PROGRAM MAIN_FBD_IL_LD //use menu "FBD/IL/LD" to switch language between FBD, IL and LD offline or online 
VAR
	Timer					: TON;
	fbFBD_IL_LD_SamplePOU 	: FB_FBD_IL_LD_SamplePOU;

	eOperation		: E_Operation := eOp_Add;
	eOperationPrev	: E_Operation := eOp_Add;
	iResultC		: DINT;
	bZero			: BOOL;
	bPos			: BOOL;
	bNeg			: BOOL;
	bTest			: BOOL;
	tTimerValue		: TIME := T#3S;
END_VAR
VAR // added by the converter: edge detectors and wires of the graphical bodies
    _w1, _w2, _w3 : ANY;
END_VAR

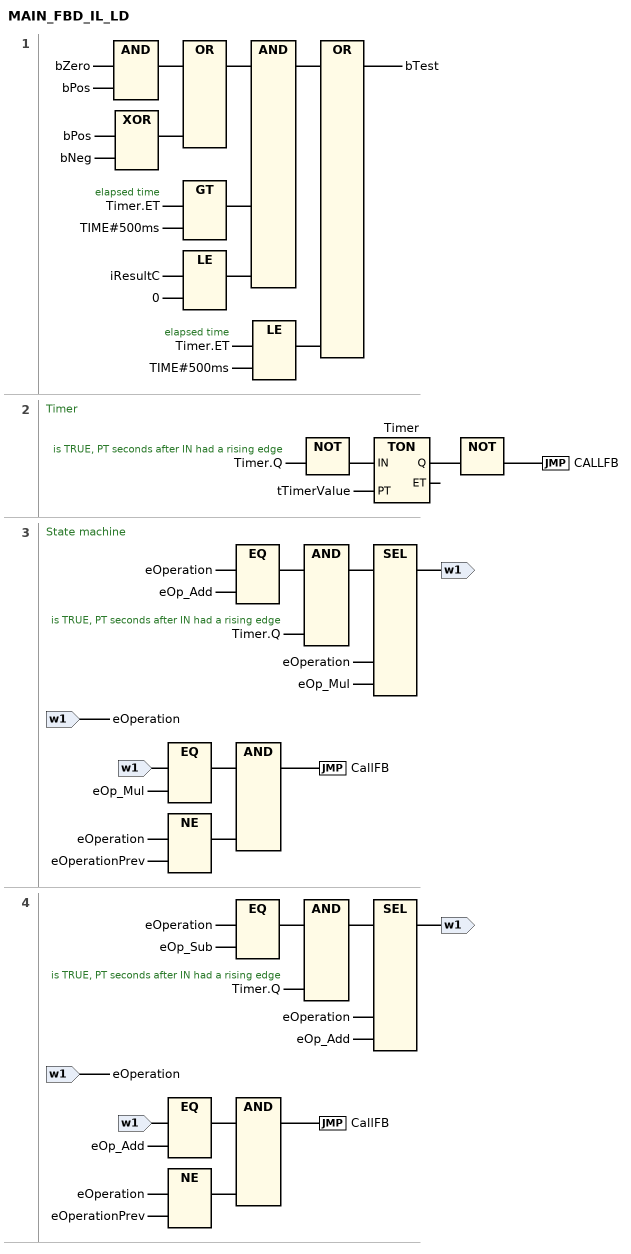
// NETWORK 1
//   Timer.ET: elapsed time
bTest := (bZero AND bPos OR bPos XOR bNeg) AND Timer.ET > TIME#500ms AND iResultC <= 0 OR Timer.ET <= TIME#500ms;

// NETWORK 2
//  Timer
//   Timer.Q: is TRUE, PT seconds after IN had a rising edge
Timer(IN := NOT Timer.Q, PT := tTimerValue); // TON
IF NOT Timer.Q THEN JMP CALLFB; END_IF

// NETWORK 3
//  State machine
//   Timer.Q: is TRUE, PT seconds after IN had a rising edge
_w1 := SEL(eOperation = eOp_Add AND Timer.Q, eOperation, eOp_Mul);
eOperation := _w1;
IF _w1 = eOp_Mul AND eOperation <> eOperationPrev THEN JMP CallFB; END_IF

// NETWORK 4
//   Timer.Q: is TRUE, PT seconds after IN had a rising edge
_w2 := SEL(eOperation = eOp_Sub AND Timer.Q, eOperation, eOp_Add);
eOperation := _w2;
IF _w2 = eOp_Add AND eOperation <> eOperationPrev THEN JMP CallFB; END_IF

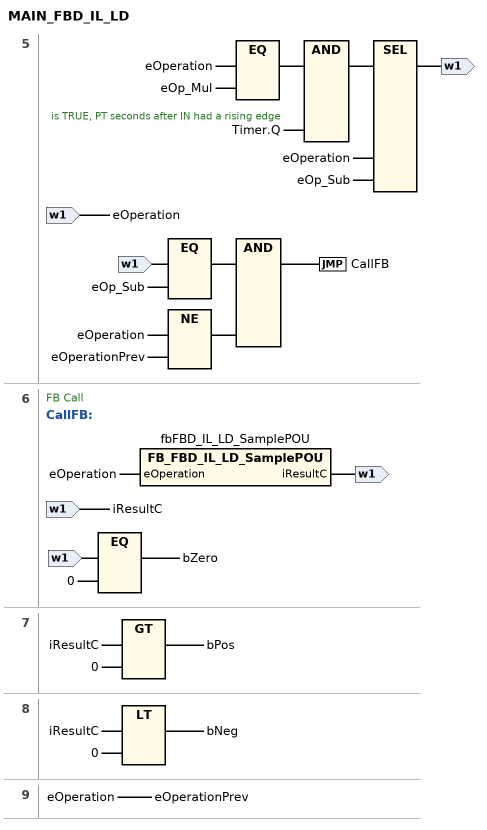
// NETWORK 5
//   Timer.Q: is TRUE, PT seconds after IN had a rising edge
_w3 := SEL(eOperation = eOp_Mul AND Timer.Q, eOperation, eOp_Sub);
eOperation := _w3;
IF _w3 = eOp_Sub AND eOperation <> eOperationPrev THEN JMP CallFB; END_IF

// NETWORK 6
//  FB Call
CallFB:
fbFBD_IL_LD_SamplePOU(eOperation := eOperation); // FB_FBD_IL_LD_SamplePOU
iResultC := fbFBD_IL_LD_SamplePOU.iResultC;
bZero := fbFBD_IL_LD_SamplePOU.iResultC = 0;

// NETWORK 7
bPos := iResultC > 0;

// NETWORK 8
bNeg := iResultC < 0;

// NETWORK 9
eOperationPrev := eOperation;

END_PROGRAM

(* stored: Version 1.1.0.1, ProductVersion 3.1.4024.11
   POU MAIN_FBD_IL_LD: Id {55328c9d-a89e-4c10-85cf-4d091864a9e8}, SpecialFunc None *)
